Omron Sysmac Studio project SPA_2 (Sysmac Studio 1.23.0.14, StandardProject)

# Controller new_Controller_0: NX1P2-1040DT1 version 1.18
Task PrimaryTask (priority 4, period or condition 2000): Programa0

VAR_GLOBAL
    Salida_0 : BOOL;  (* Salida física 0; at BuiltInIO://cpu/#0/Output_Bit_00 *)
    Salida_1 : BOOL;  (* Salida física 1; at BuiltInIO://cpu/#0/Output_Bit_01 *)
END_VAR

PROGRAM Programa0
VAR
    out_1seg : BOOL;
    cuenta : UINT;  (* Variable que contará los pulsos *)
    out1 : BOOL;
    Analog_input1 : INT;
    out9 : BOOL;
    out_9seg : BOOL;
    out_8seg : BOOL;
    out_7seg : BOOL;
    analog_input10 : REAL;
    salida : BOOL;
    sensor_11 : REAL;
    out_11 : REAL;
END_VAR
VAR_EXTERNAL
    Salida_0 : BOOL;
    Salida_1 : BOOL;
END_VAR
VAR
    _e1 : R_TRIG;
END_VAR

(* Section C7: ladder, written here as Structured Text *)

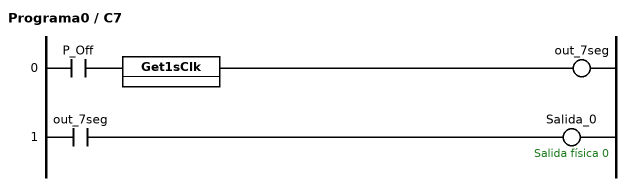
(* Rung 0 *)
out_7seg := P_Off AND Get1sClk();
(* Rung 1 *)
Salida_0 := out_7seg;

(* Section C8: ladder, written here as Structured Text *)

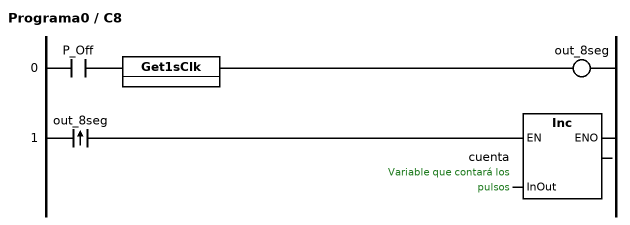
(* Rung 0 *)
out_8seg := P_Off AND Get1sClk();
(* Rung 1 *)
_e1(CLK := out_8seg);
IF _e1.Q THEN Inc(InOut := cuenta); END_IF;

(* Section C9: ladder, written here as Structured Text *)

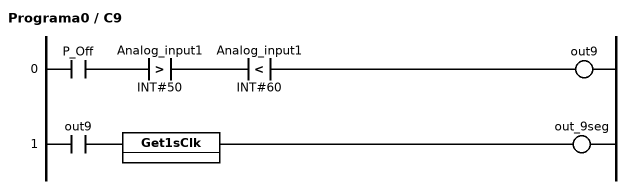
(* Rung 0 *)
out9 := P_Off AND (Analog_input1 > INT#50) AND (Analog_input1 < INT#60);
(* Rung 1 *)
out_9seg := out9 AND Get1sClk();

(* Section C10: ladder, written here as Structured Text *)

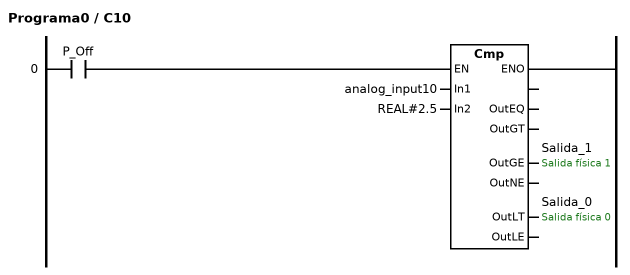
(* Rung 0 *)
IF P_Off THEN Cmp(In1 := analog_input10, In2 := REAL#2.5, OutGE => Salida_1, OutLT => Salida_0); END_IF;

(* Section C11: ladder, written here as Structured Text *)

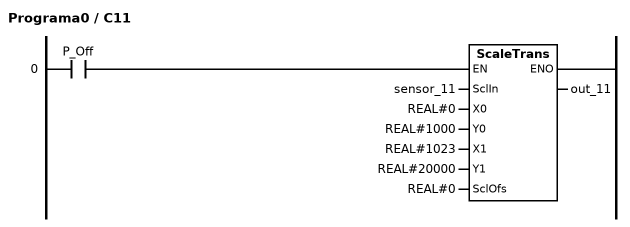
(* Rung 0 *)
IF P_Off THEN
    out_11 := ScaleTrans(SclIn := sensor_11, X0 := REAL#0, Y0 := REAL#1000, X1 := REAL#1023, Y1 := REAL#20000, SclOfs := REAL#0);
END_IF;
END_PROGRAM